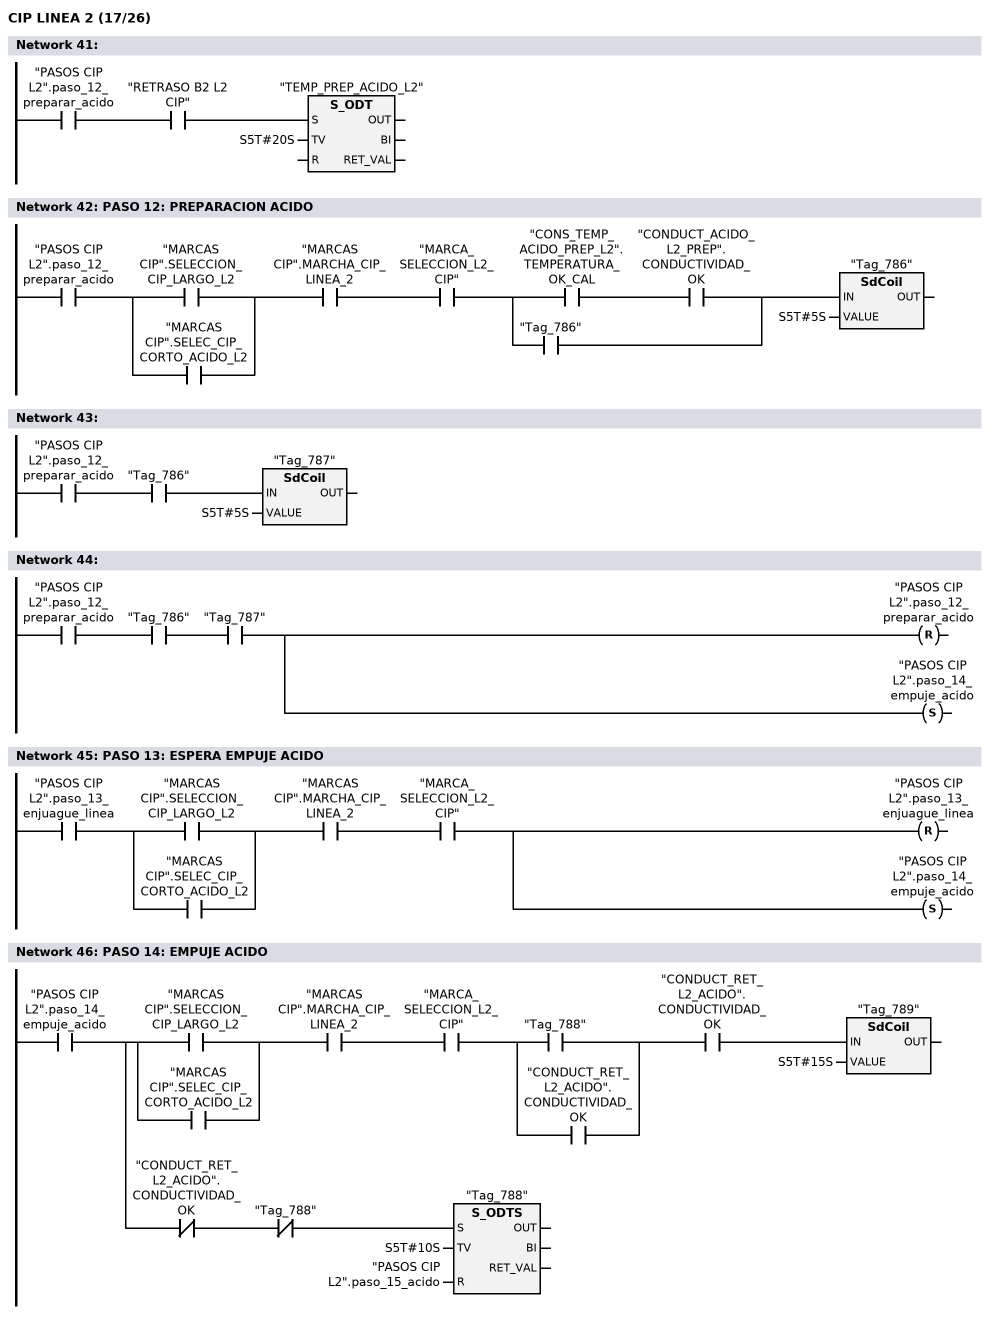
   RUNG wire#powerrail
      Contact( "PASOS CIP L2".paso_12_preparar_acido )
      Contact( "RETRASO B2 L2 CIP" )
      S_ODT(T_NO := "TEMP_PREP_ACIDO_L2", TV := S5T#20S, R :=, BI =>, RET_VAL =>)
   END_RUNG
   // the same network as SCL:
   #_s5time1 := S_ODT(T_NO := "TEMP_PREP_ACIDO_L2",
                      TV := S5T#20S,
                      S := "PASOS CIP L2".paso_12_preparar_acido AND "RETRASO B2 L2 CIP");
END_REGION

REGION Network 42: PASO 12: PREPARACION ACIDO
   // no SCL statement known for SdCoil: written as a call
   SdCoil(value := S5T#5S,
          in := "PASOS CIP L2".paso_12_preparar_acido AND ("MARCAS CIP".SELECCION_CIP_LARGO_L2 OR "MARCAS CIP".SELEC_CIP_CORTO_ACIDO_L2) AND "MARCAS CIP".MARCHA_CIP_LINEA_2 AND "MARCA_SELECCION_L2_CIP" AND (("CONS_TEMP_ACIDO_PREP_L2".TEMPERATURA_OK_CAL AND "CONDUCT_ACIDO_L2_PREP".CONDUCTIVIDAD_OK) OR "Tag_786"),
          operand := "Tag_786");
END_REGION

REGION Network 43
   // no SCL statement known for SdCoil: written as a call
   SdCoil(value := S5T#5S, operand := "Tag_787", in := "PASOS CIP L2".paso_12_preparar_acido AND "Tag_786");
END_REGION

REGION Network 44
   RUNG wire#powerrail
      Contact( "PASOS CIP L2".paso_12_preparar_acido )
      Contact( "Tag_786" )
      Contact( "Tag_787" )
      wire#w1
      R_Coil( "PASOS CIP L2".paso_12_preparar_acido )
   END_RUNG
   RUNG wire#w1
      S_Coil( "PASOS CIP L2".paso_14_empuje_acido )
   END_RUNG
   // the same network as SCL:
   #_w1 := "PASOS CIP L2".paso_12_preparar_acido AND "Tag_786" AND "Tag_787";
   IF #_w1 THEN
       "PASOS CIP L2".paso_12_preparar_acido := FALSE;
       "PASOS CIP L2".paso_14_empuje_acido := TRUE;
   END_IF;
END_REGION

REGION Network 45: PASO 13: ESPERA EMPUJE ACIDO
   RUNG wire#powerrail
      Contact( "PASOS CIP L2".paso_13_enjuague_linea )
      wire#w1
      Contact( "MARCAS CIP".SELECCION_CIP_LARGO_L2 )
      wire#w2
      Contact( "MARCAS CIP".MARCHA_CIP_LINEA_2 )
      Contact( "MARCA_SELECCION_L2_CIP" )
      wire#w3
      R_Coil( "PASOS CIP L2".paso_13_enjuague_linea )
   END_RUNG
   RUNG wire#w1
      Contact( "MARCAS CIP".SELEC_CIP_CORTO_ACIDO_L2 )
   END_RUNG wire#w2
   RUNG wire#w3
      S_Coil( "PASOS CIP L2".paso_14_empuje_acido )
   END_RUNG
   // the same network as SCL:
   #_w1 := "PASOS CIP L2".paso_13_enjuague_linea AND ("MARCAS CIP".SELECCION_CIP_LARGO_L2 OR "MARCAS CIP".SELEC_CIP_CORTO_ACIDO_L2) AND "MARCAS CIP".MARCHA_CIP_LINEA_2 AND "MARCA_SELECCION_L2_CIP";
   IF #_w1 THEN
       "PASOS CIP L2".paso_13_enjuague_linea := FALSE;
       "PASOS CIP L2".paso_14_empuje_acido := TRUE;
   END_IF;
END_REGION

REGION Network 46: PASO 14: EMPUJE ACIDO
   // no SCL statement known for SdCoil: written as a call
   #_w1 := "PASOS CIP L2".paso_14_empuje_acido;
   SdCoil(value := S5T#15S,
          operand := "Tag_789",
          in := "PASOS CIP L2".paso_14_empuje_acido AND ("MARCAS CIP".SELECCION_CIP_LARGO_L2 OR "MARCAS CIP".SELEC_CIP_CORTO_ACIDO_L2) AND "MARCAS CIP".MARCHA_CIP_LINEA_2 AND "MARCA_SELECCION_L2_CIP" AND ("Tag_788" OR "CONDUCT_RET_L2_ACIDO".CONDUCTIVIDAD_OK) AND "CONDUCT_RET_L2_ACIDO".CONDUCTIVIDAD_OK);
   #_s5time1 := S_ODTS(T_NO := "Tag_788",
                       TV := S5T#10S,
                       R := "PASOS CIP L2".paso_15_acido,
                       S := #_w1 AND NOT "CONDUCT_RET_L2_ACIDO".CONDUCTIVIDAD_OK AND NOT "Tag_788");
END_REGION

REGION Network 47
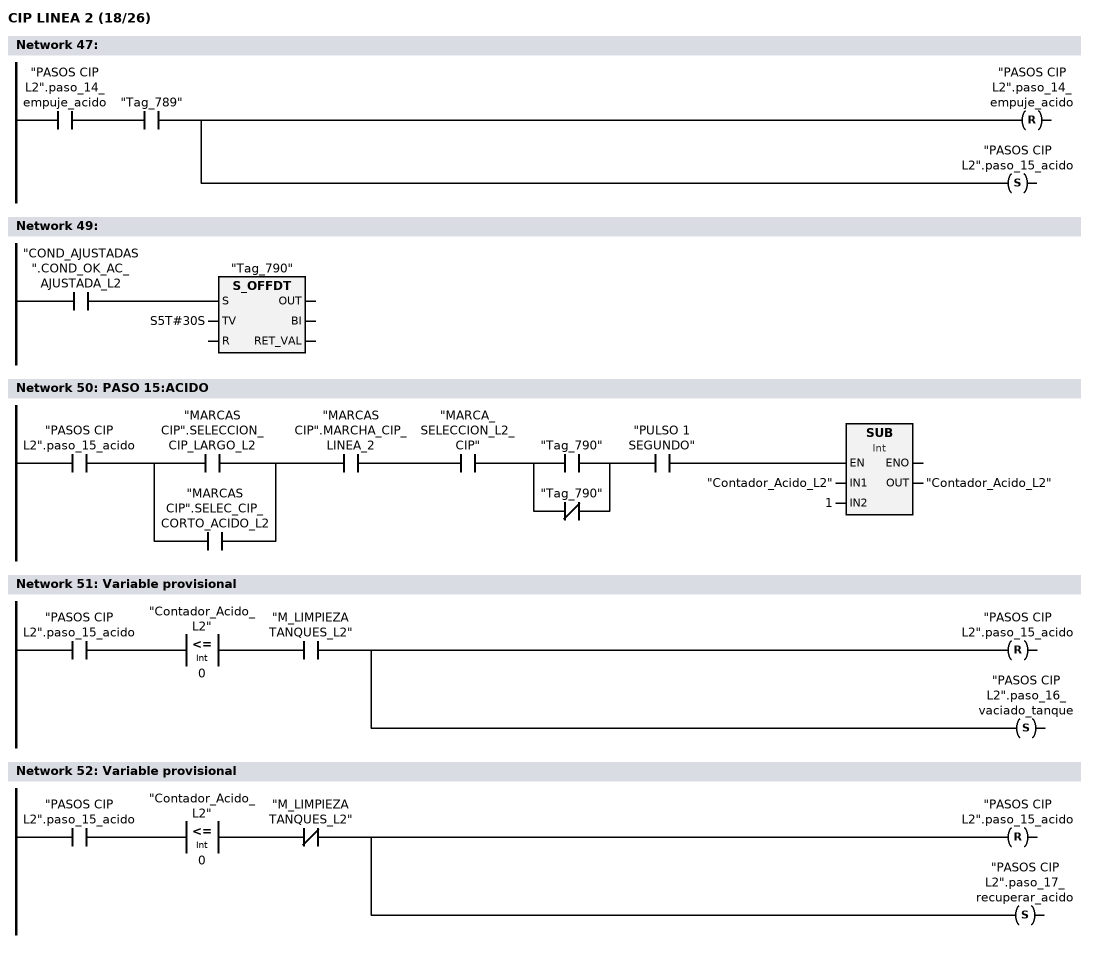
   RUNG wire#powerrail
      Contact( "PASOS CIP L2".paso_14_empuje_acido )
      Contact( "Tag_789" )
      wire#w1
      R_Coil( "PASOS CIP L2".paso_14_empuje_acido )
   END_RUNG
   RUNG wire#w1
      S_Coil( "PASOS CIP L2".paso_15_acido )
   END_RUNG
   // the same network as SCL:
   #_w1 := "PASOS CIP L2".paso_14_empuje_acido AND "Tag_789";
   IF #_w1 THEN
       "PASOS CIP L2".paso_14_empuje_acido := FALSE;
       "PASOS CIP L2".paso_15_acido := TRUE;
   END_IF;
END_REGION

NETWORK
TITLE = 
      A     "PASOS CIP L2".paso_15_acido;
      JC    c2;
      L     "SP TIM L2 CIP".TIM_PASO_15_L2;
      L     60;
      *I;
      T     "Contador_Acido_L2";
c2:   NOP   0;

REGION Network 49
   RUNG wire#powerrail
      Contact( "COND_AJUSTADAS".COND_OK_AC_AJUSTADA_L2 )
      S_OFFDT(T_NO := "Tag_790", TV := S5T#30S, R :=, BI =>, RET_VAL =>)
   END_RUNG
   // the same network as SCL:
   #_s5time1 := S_OFFDT(T_NO := "Tag_790", TV := S5T#30S, S := "COND_AJUSTADAS".COND_OK_AC_AJUSTADA_L2);
END_REGION

REGION Network 50: PASO 15:ACIDO
   RUNG wire#powerrail
      Contact( "PASOS CIP L2".paso_15_acido )
      wire#w1
      Contact( "MARCAS CIP".SELECCION_CIP_LARGO_L2 )
      wire#w2
      Contact( "MARCAS CIP".MARCHA_CIP_LINEA_2 )
      Contact( "MARCA_SELECCION_L2_CIP" )
      wire#w3
      Contact( "Tag_790" )
      wire#w4
      Contact( "PULSO 1 SEGUNDO" )
      { S7_Templates := "SrcType := Int"; S7_GenerateENO := "TRUE" } Sub(in1 := "Contador_Acido_L2", in2 := 1, out => "Contador_Acido_L2")
   END_RUNG
   RUNG wire#w1
      Contact( "MARCAS CIP".SELEC_CIP_CORTO_ACIDO_L2 )
   END_RUNG wire#w2
   RUNG wire#w3
      I_Contact( "Tag_790" )
   END_RUNG wire#w4
   // the same network as SCL:
   IF "PASOS CIP L2".paso_15_acido AND ("MARCAS CIP".SELECCION_CIP_LARGO_L2 OR "MARCAS CIP".SELEC_CIP_CORTO_ACIDO_L2) AND "MARCAS CIP".MARCHA_CIP_LINEA_2 AND "MARCA_SELECCION_L2_CIP" AND ("Tag_790" OR NOT "Tag_790") AND "PULSO 1 SEGUNDO" THEN
       "Contador_Acido_L2" := "Contador_Acido_L2" - 1;
   END_IF;
END_REGION

REGION Network 51: Variable provisional
   RUNG wire#powerrail
      Contact( "PASOS CIP L2".paso_15_acido )
      { S7_Templates := "SrcType := Int" } LE_Contact(in1 := "Contador_Acido_L2", in2 := 0)
      Contact( "M_LIMPIEZA TANQUES_L2" )
      wire#w1
      R_Coil( "PASOS CIP L2".paso_15_acido )
   END_RUNG
   RUNG wire#w1
      S_Coil( "PASOS CIP L2".paso_16_vaciado_tanque )
   END_RUNG
   // the same network as SCL:
   #_w1 := "PASOS CIP L2".paso_15_acido AND ("Contador_Acido_L2" <= 0) AND "M_LIMPIEZA TANQUES_L2";
   IF #_w1 THEN
       "PASOS CIP L2".paso_15_acido := FALSE;
       "PASOS CIP L2".paso_16_vaciado_tanque := TRUE;
   END_IF;
END_REGION

REGION Network 52: Variable provisional
   RUNG wire#powerrail
      Contact( "PASOS CIP L2".paso_15_acido )
      { S7_Templates := "SrcType := Int" } LE_Contact(in1 := "Contador_Acido_L2", in2 := 0)
      I_Contact( "M_LIMPIEZA TANQUES_L2" )
      wire#w1
      R_Coil( "PASOS CIP L2".paso_15_acido )
   END_RUNG
   RUNG wire#w1
      S_Coil( "PASOS CIP L2".paso_17_recuperar_acido )
   END_RUNG
   // the same network as SCL:
   #_w1 := "PASOS CIP L2".paso_15_acido AND ("Contador_Acido_L2" <= 0) AND NOT "M_LIMPIEZA TANQUES_L2";
   IF #_w1 THEN
       "PASOS CIP L2".paso_15_acido := FALSE;
       "PASOS CIP L2".paso_17_recuperar_acido := TRUE;
   END_IF;
END_REGION

REGION Network 53: PASO 16: VACIADO SI TANQUES
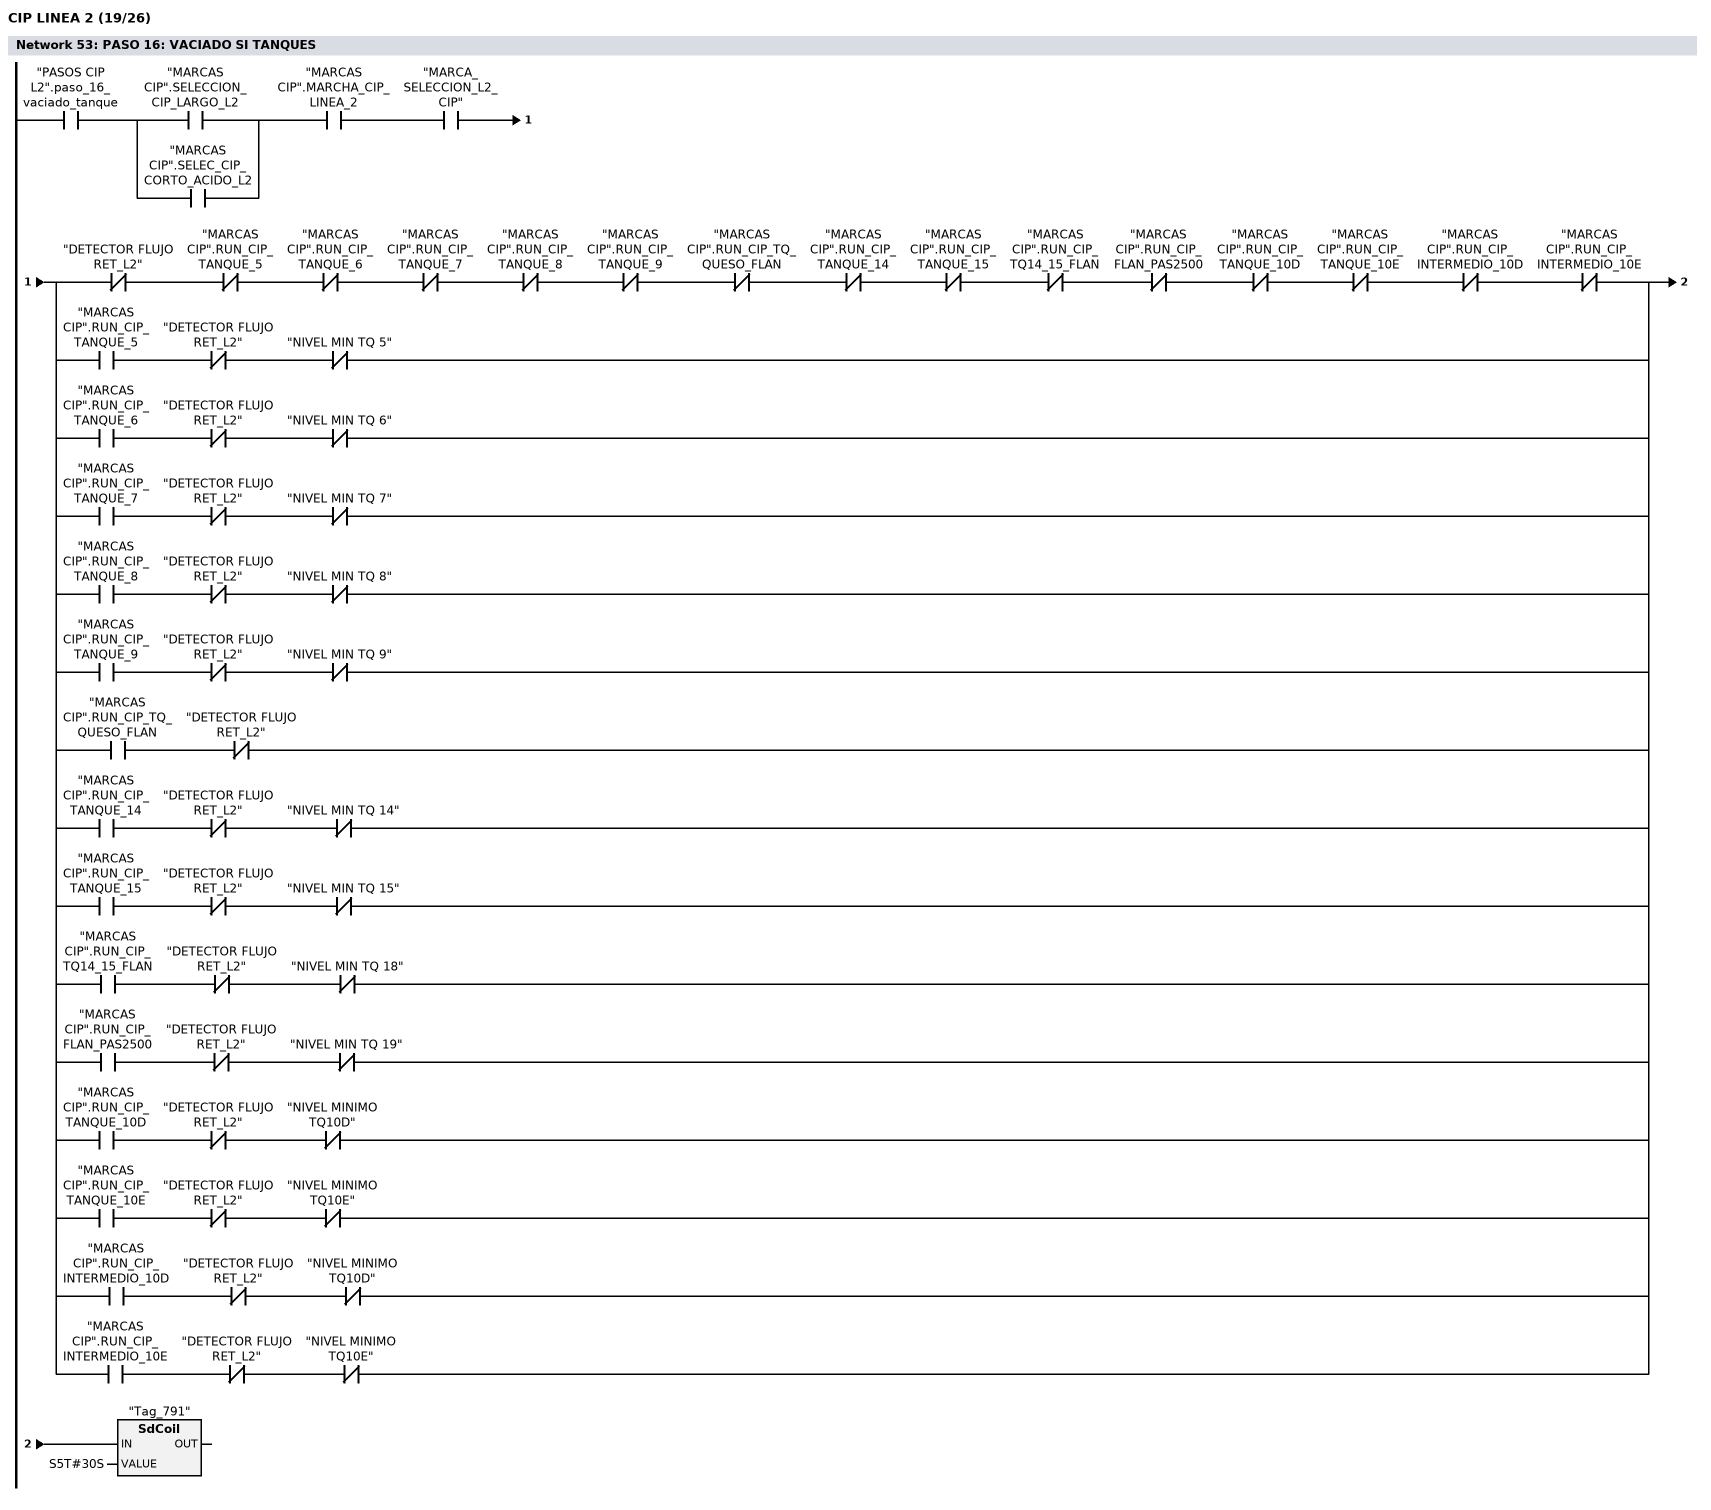
   // no SCL statement known for SdCoil: written as a call
   SdCoil(value := S5T#30S,
          in := "PASOS CIP L2".paso_16_vaciado_tanque AND ("MARCAS CIP".SELECCION_CIP_LARGO_L2 OR "MARCAS CIP".SELEC_CIP_CORTO_ACIDO_L2) AND "MARCAS CIP".MARCHA_CIP_LINEA_2 AND "MARCA_SELECCION_L2_CIP" AND ((NOT "DETECTOR FLUJO RET_L2" AND NOT "MARCAS CIP".RUN_CIP_TANQUE_5 AND NOT "MARCAS CIP".RUN_CIP_TANQUE_6 AND NOT "MARCAS CIP".RUN_CIP_TANQUE_7 AND NOT "MARCAS CIP".RUN_CIP_TANQUE_8 AND NOT "MARCAS CIP".RUN_CIP_TANQUE_9 AND NOT "MARCAS CIP".RUN_CIP_TQ_QUESO_FLAN AND NOT "MARCAS CIP".RUN_CIP_TANQUE_14 AND NOT "MARCAS CIP".RUN_CIP_TANQUE_15 AND NOT "MARCAS CIP".RUN_CIP_TQ14_15_FLAN AND NOT "MARCAS CIP".RUN_CIP_FLAN_PAS2500 AND NOT "MARCAS CIP".RUN_CIP_TANQUE_10D AND NOT "MARCAS CIP".RUN_CIP_TANQUE_10E AND NOT "MARCAS CIP".RUN_CIP_INTERMEDIO_10D AND NOT "MARCAS CIP".RUN_CIP_INTERMEDIO_10E) OR ("MARCAS CIP".RUN_CIP_TANQUE_5 AND NOT "DETECTOR FLUJO RET_L2" AND NOT "NIVEL MIN TQ 5") OR ("MARCAS CIP".RUN_CIP_TANQUE_6 AND NOT "DETECTOR FLUJO RET_L2" AND NOT "NIVEL MIN TQ 6") OR ("MARCAS CIP".RUN_CIP_TANQUE_7 AND NOT "DETECTOR FLUJO RET_L2" AND NOT "NIVEL MIN TQ 7") OR ("MARCAS CIP".RUN_CIP_TANQUE_8 AND NOT "DETECTOR FLUJO RET_L2" AND NOT "NIVEL MIN TQ 8") OR ("MARCAS CIP".RUN_CIP_TANQUE_9 AND NOT "DETECTOR FLUJO RET_L2" AND NOT "NIVEL MIN TQ 9") OR ("MARCAS CIP".RUN_CIP_TQ_QUESO_FLAN AND NOT "DETECTOR FLUJO RET_L2") OR ("MARCAS CIP".RUN_CIP_TANQUE_14 AND NOT "DETECTOR FLUJO RET_L2" AND NOT "NIVEL MIN TQ 14") OR ("MARCAS CIP".RUN_CIP_TANQUE_15 AND NOT "DETECTOR FLUJO RET_L2" AND NOT "NIVEL MIN TQ 15") OR ("MARCAS CIP".RUN_CIP_TQ14_15_FLAN AND NOT "DETECTOR FLUJO RET_L2" AND NOT "NIVEL MIN TQ 18") OR ("MARCAS CIP".RUN_CIP_FLAN_PAS2500 AND NOT "DETECTOR FLUJO RET_L2" AND NOT "NIVEL MIN TQ 19") OR ("MARCAS CIP".RUN_CIP_TANQUE_10D AND NOT "DETECTOR FLUJO RET_L2" AND NOT "NIVEL MINIMO TQ10D") OR ("MARCAS CIP".RUN_CIP_TANQUE_10E AND NOT "DETECTOR FLUJO RET_L2" AND NOT "NIVEL MINIMO TQ10E") OR ("MARCAS CIP".RUN_CIP_INTERMEDIO_10D AND NOT "DETECTOR FLUJO RET_L2" AND NOT "NIVEL MINIMO TQ10D") OR ("MARCAS CIP".RUN_CIP_INTERMEDIO_10E AND NOT "DETECTOR FLUJO RET_L2" AND NOT "NIVEL MINIMO TQ10E")),
          operand := "Tag_791");
END_REGION

REGION Network 54: Variable provisional
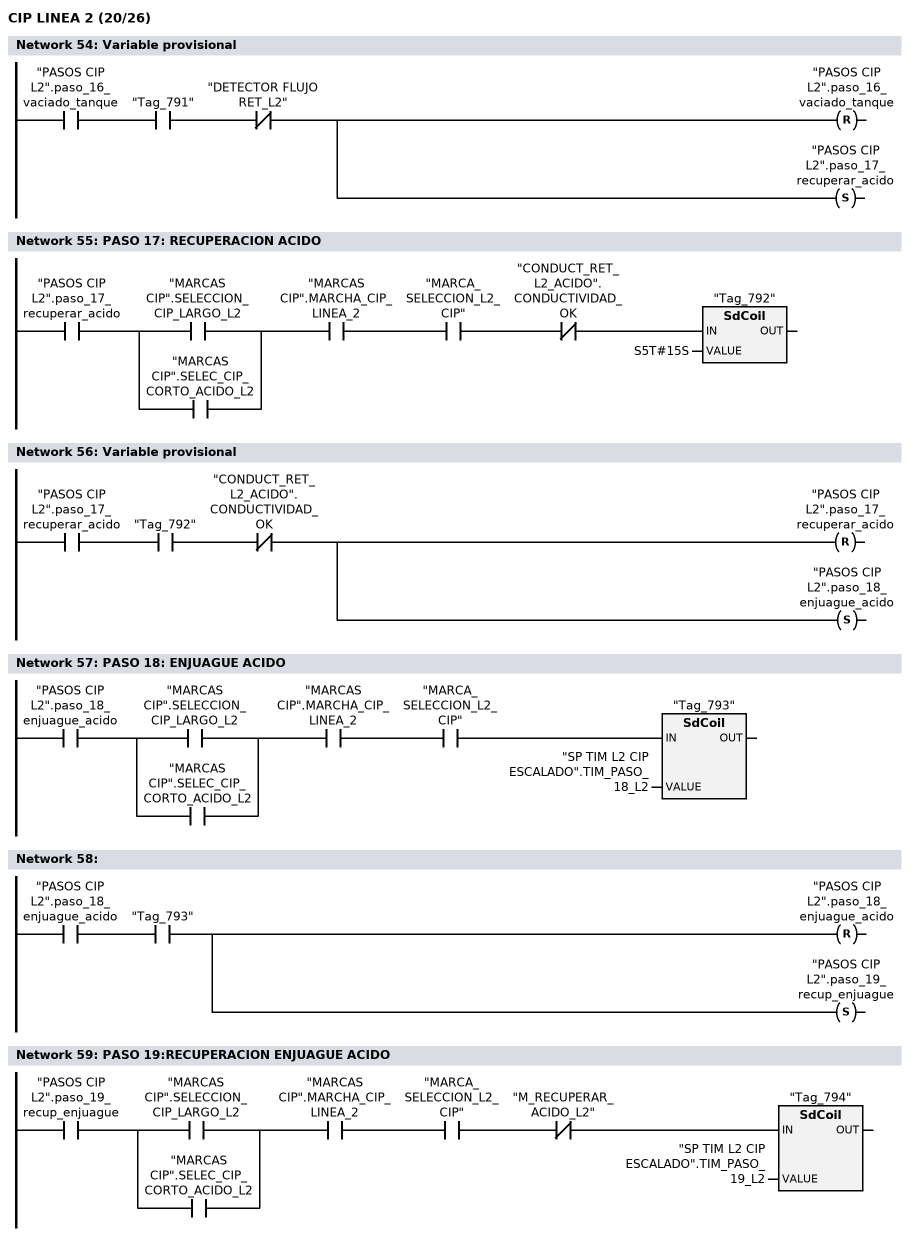
   RUNG wire#powerrail
      Contact( "PASOS CIP L2".paso_16_vaciado_tanque )
      Contact( "Tag_791" )
      I_Contact( "DETECTOR FLUJO RET_L2" )
      wire#w1
      R_Coil( "PASOS CIP L2".paso_16_vaciado_tanque )
   END_RUNG
   RUNG wire#w1
      S_Coil( "PASOS CIP L2".paso_17_recuperar_acido )
   END_RUNG
   // the same network as SCL:
   #_w1 := "PASOS CIP L2".paso_16_vaciado_tanque AND "Tag_791" AND NOT "DETECTOR FLUJO RET_L2";
   IF #_w1 THEN
       "PASOS CIP L2".paso_16_vaciado_tanque := FALSE;
       "PASOS CIP L2".paso_17_recuperar_acido := TRUE;
   END_IF;
END_REGION

REGION Network 55: PASO 17: RECUPERACION ACIDO
   // no SCL statement known for SdCoil: written as a call
   SdCoil(value := S5T#15S,
          operand := "Tag_792",
          in := "PASOS CIP L2".paso_17_recuperar_acido AND ("MARCAS CIP".SELECCION_CIP_LARGO_L2 OR "MARCAS CIP".SELEC_CIP_CORTO_ACIDO_L2) AND "MARCAS CIP".MARCHA_CIP_LINEA_2 AND "MARCA_SELECCION_L2_CIP" AND NOT "CONDUCT_RET_L2_ACIDO".CONDUCTIVIDAD_OK);
END_REGION

REGION Network 56: Variable provisional
   RUNG wire#powerrail
      Contact( "PASOS CIP L2".paso_17_recuperar_acido )
      Contact( "Tag_792" )
      I_Contact( "CONDUCT_RET_L2_ACIDO".CONDUCTIVIDAD_OK )
      wire#w1
      R_Coil( "PASOS CIP L2".paso_17_recuperar_acido )
   END_RUNG
   RUNG wire#w1
      S_Coil( "PASOS CIP L2".paso_18_enjuague_acido )
   END_RUNG
   // the same network as SCL:
   #_w1 := "PASOS CIP L2".paso_17_recuperar_acido AND "Tag_792" AND NOT "CONDUCT_RET_L2_ACIDO".CONDUCTIVIDAD_OK;
   IF #_w1 THEN
       "PASOS CIP L2".paso_17_recuperar_acido := FALSE;
       "PASOS CIP L2".paso_18_enjuague_acido := TRUE;
   END_IF;
END_REGION

REGION Network 57: PASO 18: ENJUAGUE ACIDO
   // no SCL statement known for SdCoil: written as a call
   SdCoil(value := "SP TIM L2 CIP ESCALADO".TIM_PASO_18_L2,
          operand := "Tag_793",
          in := "PASOS CIP L2".paso_18_enjuague_acido AND ("MARCAS CIP".SELECCION_CIP_LARGO_L2 OR "MARCAS CIP".SELEC_CIP_CORTO_ACIDO_L2) AND "MARCAS CIP".MARCHA_CIP_LINEA_2 AND "MARCA_SELECCION_L2_CIP");
END_REGION

REGION Network 58
   RUNG wire#powerrail
      Contact( "PASOS CIP L2".paso_18_enjuague_acido )
      Contact( "Tag_793" )
      wire#w1
      R_Coil( "PASOS CIP L2".paso_18_enjuague_acido )
   END_RUNG
   RUNG wire#w1
      S_Coil( "PASOS CIP L2".paso_19_recup_enjuague )
   END_RUNG
   // the same network as SCL:
   #_w1 := "PASOS CIP L2".paso_18_enjuague_acido AND "Tag_793";
   IF #_w1 THEN
       "PASOS CIP L2".paso_18_enjuague_acido := FALSE;
       "PASOS CIP L2".paso_19_recup_enjuague := TRUE;
   END_IF;
END_REGION

REGION Network 59: PASO 19:RECUPERACION ENJUAGUE ACIDO
   // no SCL statement known for SdCoil: written as a call
   SdCoil(value := "SP TIM L2 CIP ESCALADO".TIM_PASO_19_L2,
          operand := "Tag_794",
          in := "PASOS CIP L2".paso_19_recup_enjuague AND ("MARCAS CIP".SELECCION_CIP_LARGO_L2 OR "MARCAS CIP".SELEC_CIP_CORTO_ACIDO_L2) AND "MARCAS CIP".MARCHA_CIP_LINEA_2 AND "MARCA_SELECCION_L2_CIP" AND NOT "M_RECUPERAR_ACIDO_L2");
END_REGION

REGION Network 60
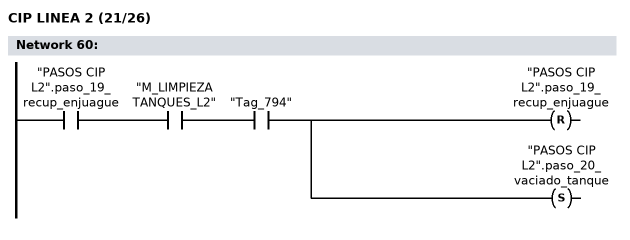
   RUNG wire#powerrail
      Contact( "PASOS CIP L2".paso_19_recup_enjuague )
      Contact( "M_LIMPIEZA TANQUES_L2" )
      Contact( "Tag_794" )
      wire#w1
      R_Coil( "PASOS CIP L2".paso_19_recup_enjuague )
   END_RUNG
   RUNG wire#w1
      S_Coil( "PASOS CIP L2".paso_20_vaciado_tanque )
   END_RUNG
   // the same network as SCL:
   #_w1 := "PASOS CIP L2".paso_19_recup_enjuague AND "M_LIMPIEZA TANQUES_L2" AND "Tag_794";
   IF #_w1 THEN
       "PASOS CIP L2".paso_19_recup_enjuague := FALSE;
       "PASOS CIP L2".paso_20_vaciado_tanque := TRUE;
   END_IF;
END_REGION

REGION Network 61
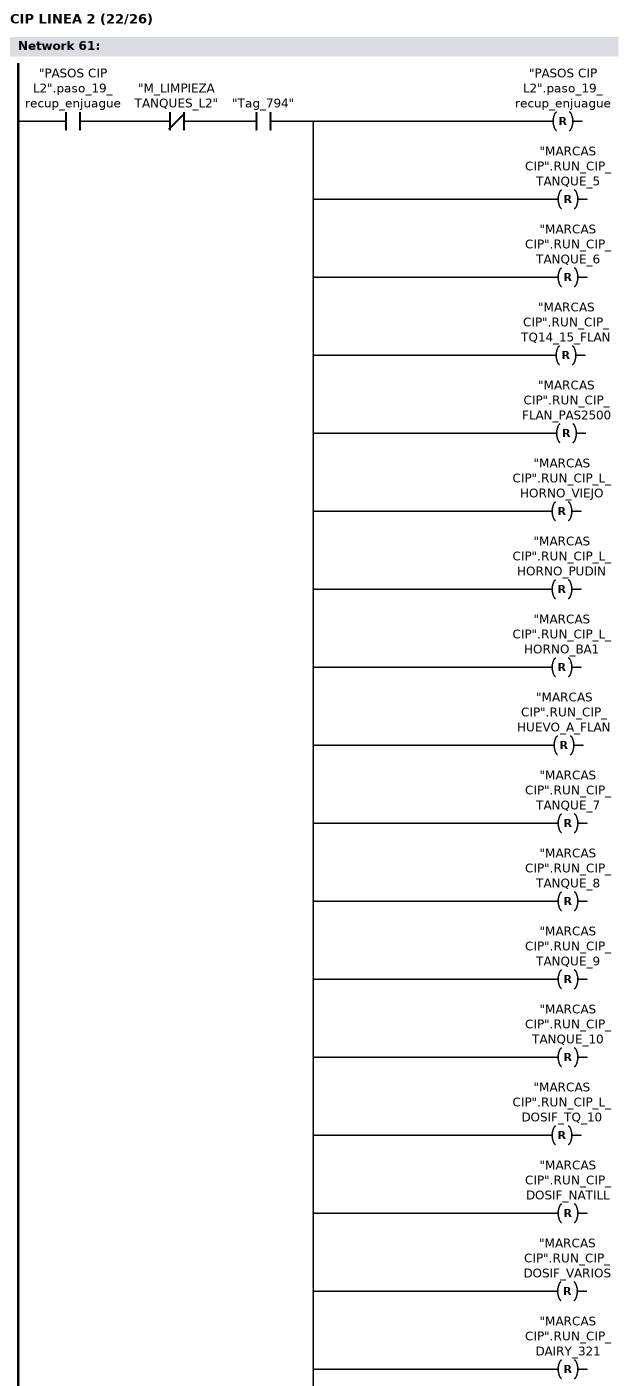
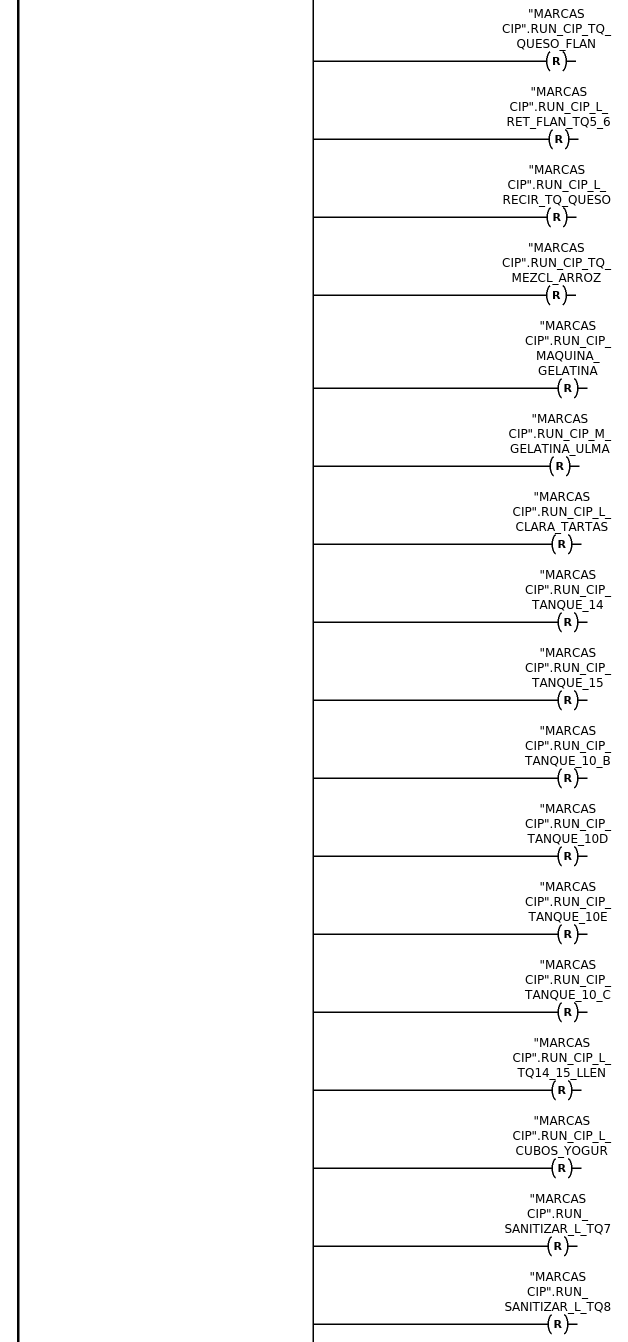
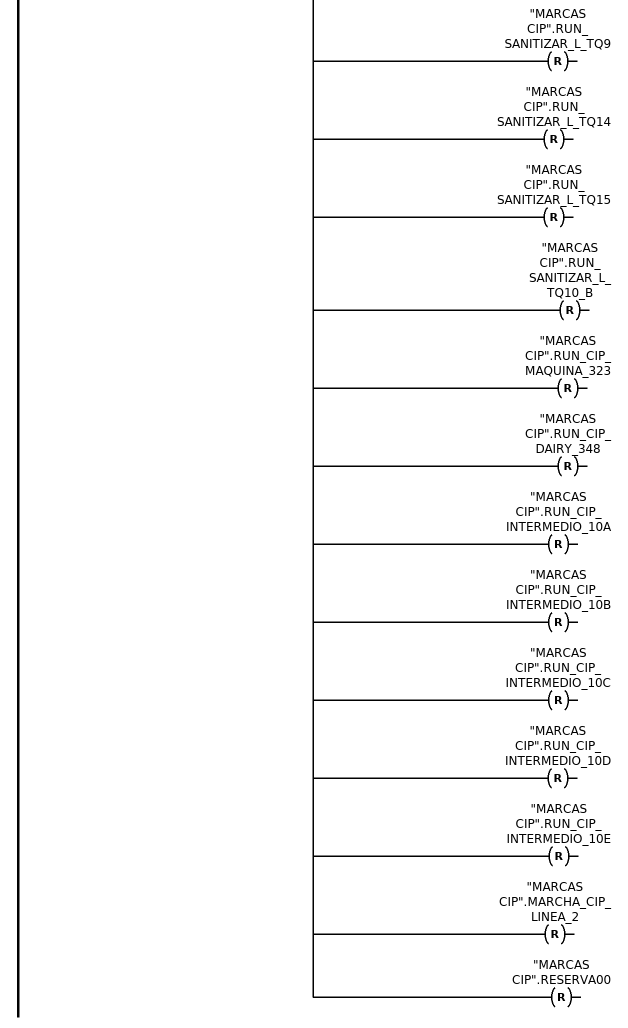
   RUNG wire#powerrail
      Contact( "PASOS CIP L2".paso_19_recup_enjuague )
      I_Contact( "M_LIMPIEZA TANQUES_L2" )
      Contact( "Tag_794" )
      wire#w1
      R_Coil( "PASOS CIP L2".paso_19_recup_enjuague )
   END_RUNG
   RUNG wire#w1
      R_Coil( "MARCAS CIP".RUN_CIP_TANQUE_5 )
   END_RUNG
   RUNG wire#w1
      R_Coil( "MARCAS CIP".RUN_CIP_TANQUE_6 )
   END_RUNG
   RUNG wire#w1
      R_Coil( "MARCAS CIP".RUN_CIP_TQ14_15_FLAN )
   END_RUNG
   RUNG wire#w1
      R_Coil( "MARCAS CIP".RUN_CIP_FLAN_PAS2500 )
   END_RUNG
   RUNG wire#w1
      R_Coil( "MARCAS CIP".RUN_CIP_L_HORNO_VIEJO )
   END_RUNG
   RUNG wire#w1
      R_Coil( "MARCAS CIP".RUN_CIP_L_HORNO_PUDIN )
   END_RUNG
   RUNG wire#w1
      R_Coil( "MARCAS CIP".RUN_CIP_L_HORNO_BA1 )
   END_RUNG
   RUNG wire#w1
      R_Coil( "MARCAS CIP".RUN_CIP_HUEVO_A_FLAN )
   END_RUNG
   RUNG wire#w1
      R_Coil( "MARCAS CIP".RUN_CIP_TANQUE_7 )
   END_RUNG
   RUNG wire#w1
      R_Coil( "MARCAS CIP".RUN_CIP_TANQUE_8 )
   END_RUNG
   RUNG wire#w1
      R_Coil( "MARCAS CIP".RUN_CIP_TANQUE_9 )
   END_RUNG
   RUNG wire#w1
      R_Coil( "MARCAS CIP".RUN_CIP_TANQUE_10 )
   END_RUNG
   RUNG wire#w1
      R_Coil( "MARCAS CIP".RUN_CIP_L_DOSIF_TQ_10 )
   END_RUNG
   RUNG wire#w1
      R_Coil( "MARCAS CIP".RUN_CIP_DOSIF_NATILL )
   END_RUNG
   RUNG wire#w1
      R_Coil( "MARCAS CIP".RUN_CIP_DOSIF_VARIOS )
   END_RUNG
   RUNG wire#w1
      R_Coil( "MARCAS CIP".RUN_CIP_DAIRY_321 )
   END_RUNG
   RUNG wire#w1
      R_Coil( "MARCAS CIP".RUN_CIP_TQ_QUESO_FLAN )
   END_RUNG
   RUNG wire#w1
      R_Coil( "MARCAS CIP".RUN_CIP_L_RET_FLAN_TQ5_6 )
   END_RUNG
   RUNG wire#w1
      R_Coil( "MARCAS CIP".RUN_CIP_L_RECIR_TQ_QUESO )
   END_RUNG
   RUNG wire#w1
      R_Coil( "MARCAS CIP".RUN_CIP_TQ_MEZCL_ARROZ )
   END_RUNG
   RUNG wire#w1
      R_Coil( "MARCAS CIP".RUN_CIP_MAQUINA_GELATINA )
   END_RUNG
   RUNG wire#w1
      R_Coil( "MARCAS CIP".RUN_CIP_M_GELATINA_ULMA )
   END_RUNG
   RUNG wire#w1
      R_Coil( "MARCAS CIP".RUN_CIP_L_CLARA_TARTAS )
   END_RUNG
   RUNG wire#w1
      R_Coil( "MARCAS CIP".RUN_CIP_TANQUE_14 )
   END_RUNG
   RUNG wire#w1
      R_Coil( "MARCAS CIP".RUN_CIP_TANQUE_15 )
   END_RUNG
   RUNG wire#w1
      R_Coil( "MARCAS CIP".RUN_CIP_TANQUE_10_B )
   END_RUNG
   RUNG wire#w1
      R_Coil( "MARCAS CIP".RUN_CIP_TANQUE_10D )
   END_RUNG
   RUNG wire#w1
      R_Coil( "MARCAS CIP".RUN_CIP_TANQUE_10E )
   END_RUNG
   RUNG wire#w1
      R_Coil( "MARCAS CIP".RUN_CIP_TANQUE_10_C )
   END_RUNG
   RUNG wire#w1
      R_Coil( "MARCAS CIP".RUN_CIP_L_TQ14_15_LLEN )
   END_RUNG
   RUNG wire#w1
      R_Coil( "MARCAS CIP".RUN_CIP_L_CUBOS_YOGUR )
   END_RUNG
   RUNG wire#w1
      R_Coil( "MARCAS CIP".RUN_SANITIZAR_L_TQ7 )
   END_RUNG
   RUNG wire#w1
      R_Coil( "MARCAS CIP".RUN_SANITIZAR_L_TQ8 )
   END_RUNG
   RUNG wire#w1
      R_Coil( "MARCAS CIP".RUN_SANITIZAR_L_TQ9 )
   END_RUNG
   RUNG wire#w1
      R_Coil( "MARCAS CIP".RUN_SANITIZAR_L_TQ14 )
   END_RUNG
   RUNG wire#w1
      R_Coil( "MARCAS CIP".RUN_SANITIZAR_L_TQ15 )
   END_RUNG
   RUNG wire#w1
      R_Coil( "MARCAS CIP".RUN_SANITIZAR_L_TQ10_B )
   END_RUNG
   RUNG wire#w1
      R_Coil( "MARCAS CIP".RUN_CIP_MAQUINA_323 )
   END_RUNG
   RUNG wire#w1
      R_Coil( "MARCAS CIP".RUN_CIP_DAIRY_348 )
   END_RUNG
   RUNG wire#w1
      R_Coil( "MARCAS CIP".RUN_CIP_INTERMEDIO_10A )
   END_RUNG
   RUNG wire#w1
      R_Coil( "MARCAS CIP".RUN_CIP_INTERMEDIO_10B )
   END_RUNG
   RUNG wire#w1
      R_Coil( "MARCAS CIP".RUN_CIP_INTERMEDIO_10C )
   END_RUNG
   RUNG wire#w1
      R_Coil( "MARCAS CIP".RUN_CIP_INTERMEDIO_10D )
   END_RUNG
   RUNG wire#w1
      R_Coil( "MARCAS CIP".RUN_CIP_INTERMEDIO_10E )
   END_RUNG
   RUNG wire#w1
      R_Coil( "MARCAS CIP".MARCHA_CIP_LINEA_2 )
   END_RUNG
   RUNG wire#w1
      R_Coil( "MARCAS CIP".RESERVA00 )
   END_RUNG
   // the same network as SCL:
   #_w1 := "PASOS CIP L2".paso_19_recup_enjuague AND NOT "M_LIMPIEZA TANQUES_L2" AND "Tag_794";
   IF #_w1 THEN
       "PASOS CIP L2".paso_19_recup_enjuague := FALSE;
       "MARCAS CIP".RUN_CIP_TANQUE_5 := FALSE;
       "MARCAS CIP".RUN_CIP_TANQUE_6 := FALSE;
       "MARCAS CIP".RUN_CIP_TQ14_15_FLAN := FALSE;
       "MARCAS CIP".RUN_CIP_FLAN_PAS2500 := FALSE;
       "MARCAS CIP".RUN_CIP_L_HORNO_VIEJO := FALSE;
       "MARCAS CIP".RUN_CIP_L_HORNO_PUDIN := FALSE;
       "MARCAS CIP".RUN_CIP_L_HORNO_BA1 := FALSE;
       "MARCAS CIP".RUN_CIP_HUEVO_A_FLAN := FALSE;
       "MARCAS CIP".RUN_CIP_TANQUE_7 := FALSE;
       "MARCAS CIP".RUN_CIP_TANQUE_8 := FALSE;
       "MARCAS CIP".RUN_CIP_TANQUE_9 := FALSE;
       "MARCAS CIP".RUN_CIP_TANQUE_10 := FALSE;
       "MARCAS CIP".RUN_CIP_L_DOSIF_TQ_10 := FALSE;
       "MARCAS CIP".RUN_CIP_DOSIF_NATILL := FALSE;
       "MARCAS CIP".RUN_CIP_DOSIF_VARIOS := FALSE;
       "MARCAS CIP".RUN_CIP_DAIRY_321 := FALSE;
       "MARCAS CIP".RUN_CIP_TQ_QUESO_FLAN := FALSE;
       "MARCAS CIP".RUN_CIP_L_RET_FLAN_TQ5_6 := FALSE;
       "MARCAS CIP".RUN_CIP_L_RECIR_TQ_QUESO := FALSE;
       "MARCAS CIP".RUN_CIP_TQ_MEZCL_ARROZ := FALSE;
       "MARCAS CIP".RUN_CIP_MAQUINA_GELATINA := FALSE;
       "MARCAS CIP".RUN_CIP_M_GELATINA_ULMA := FALSE;
       "MARCAS CIP".RUN_CIP_L_CLARA_TARTAS := FALSE;
       "MARCAS CIP".RUN_CIP_TANQUE_14 := FALSE;
       "MARCAS CIP".RUN_CIP_TANQUE_15 := FALSE;
       "MARCAS CIP".RUN_CIP_TANQUE_10_B := FALSE;
       "MARCAS CIP".RUN_CIP_TANQUE_10D := FALSE;
       "MARCAS CIP".RUN_CIP_TANQUE_10E := FALSE;
       "MARCAS CIP".RUN_CIP_TANQUE_10_C := FALSE;
       "MARCAS CIP".RUN_CIP_L_TQ14_15_LLEN := FALSE;
       "MARCAS CIP".RUN_CIP_L_CUBOS_YOGUR := FALSE;
       "MARCAS CIP".RUN_SANITIZAR_L_TQ7 := FALSE;
       "MARCAS CIP".RUN_SANITIZAR_L_TQ8 := FALSE;
       "MARCAS CIP".RUN_SANITIZAR_L_TQ9 := FALSE;
       "MARCAS CIP".RUN_SANITIZAR_L_TQ14 := FALSE;
       "MARCAS CIP".RUN_SANITIZAR_L_TQ15 := FALSE;
       "MARCAS CIP".RUN_SANITIZAR_L_TQ10_B := FALSE;
       "MARCAS CIP".RUN_CIP_MAQUINA_323 := FALSE;
       "MARCAS CIP".RUN_CIP_DAIRY_348 := FALSE;
       "MARCAS CIP".RUN_CIP_INTERMEDIO_10A := FALSE;
       "MARCAS CIP".RUN_CIP_INTERMEDIO_10B := FALSE;
       "MARCAS CIP".RUN_CIP_INTERMEDIO_10C := FALSE;
       "MARCAS CIP".RUN_CIP_INTERMEDIO_10D := FALSE;
       "MARCAS CIP".RUN_CIP_INTERMEDIO_10E := FALSE;
       "MARCAS CIP".MARCHA_CIP_LINEA_2 := FALSE;
       "MARCAS CIP".RESERVA00 := FALSE;
   END_IF;
END_REGION

REGION Network 62: PASO 19: VACIADO SI TANQUES
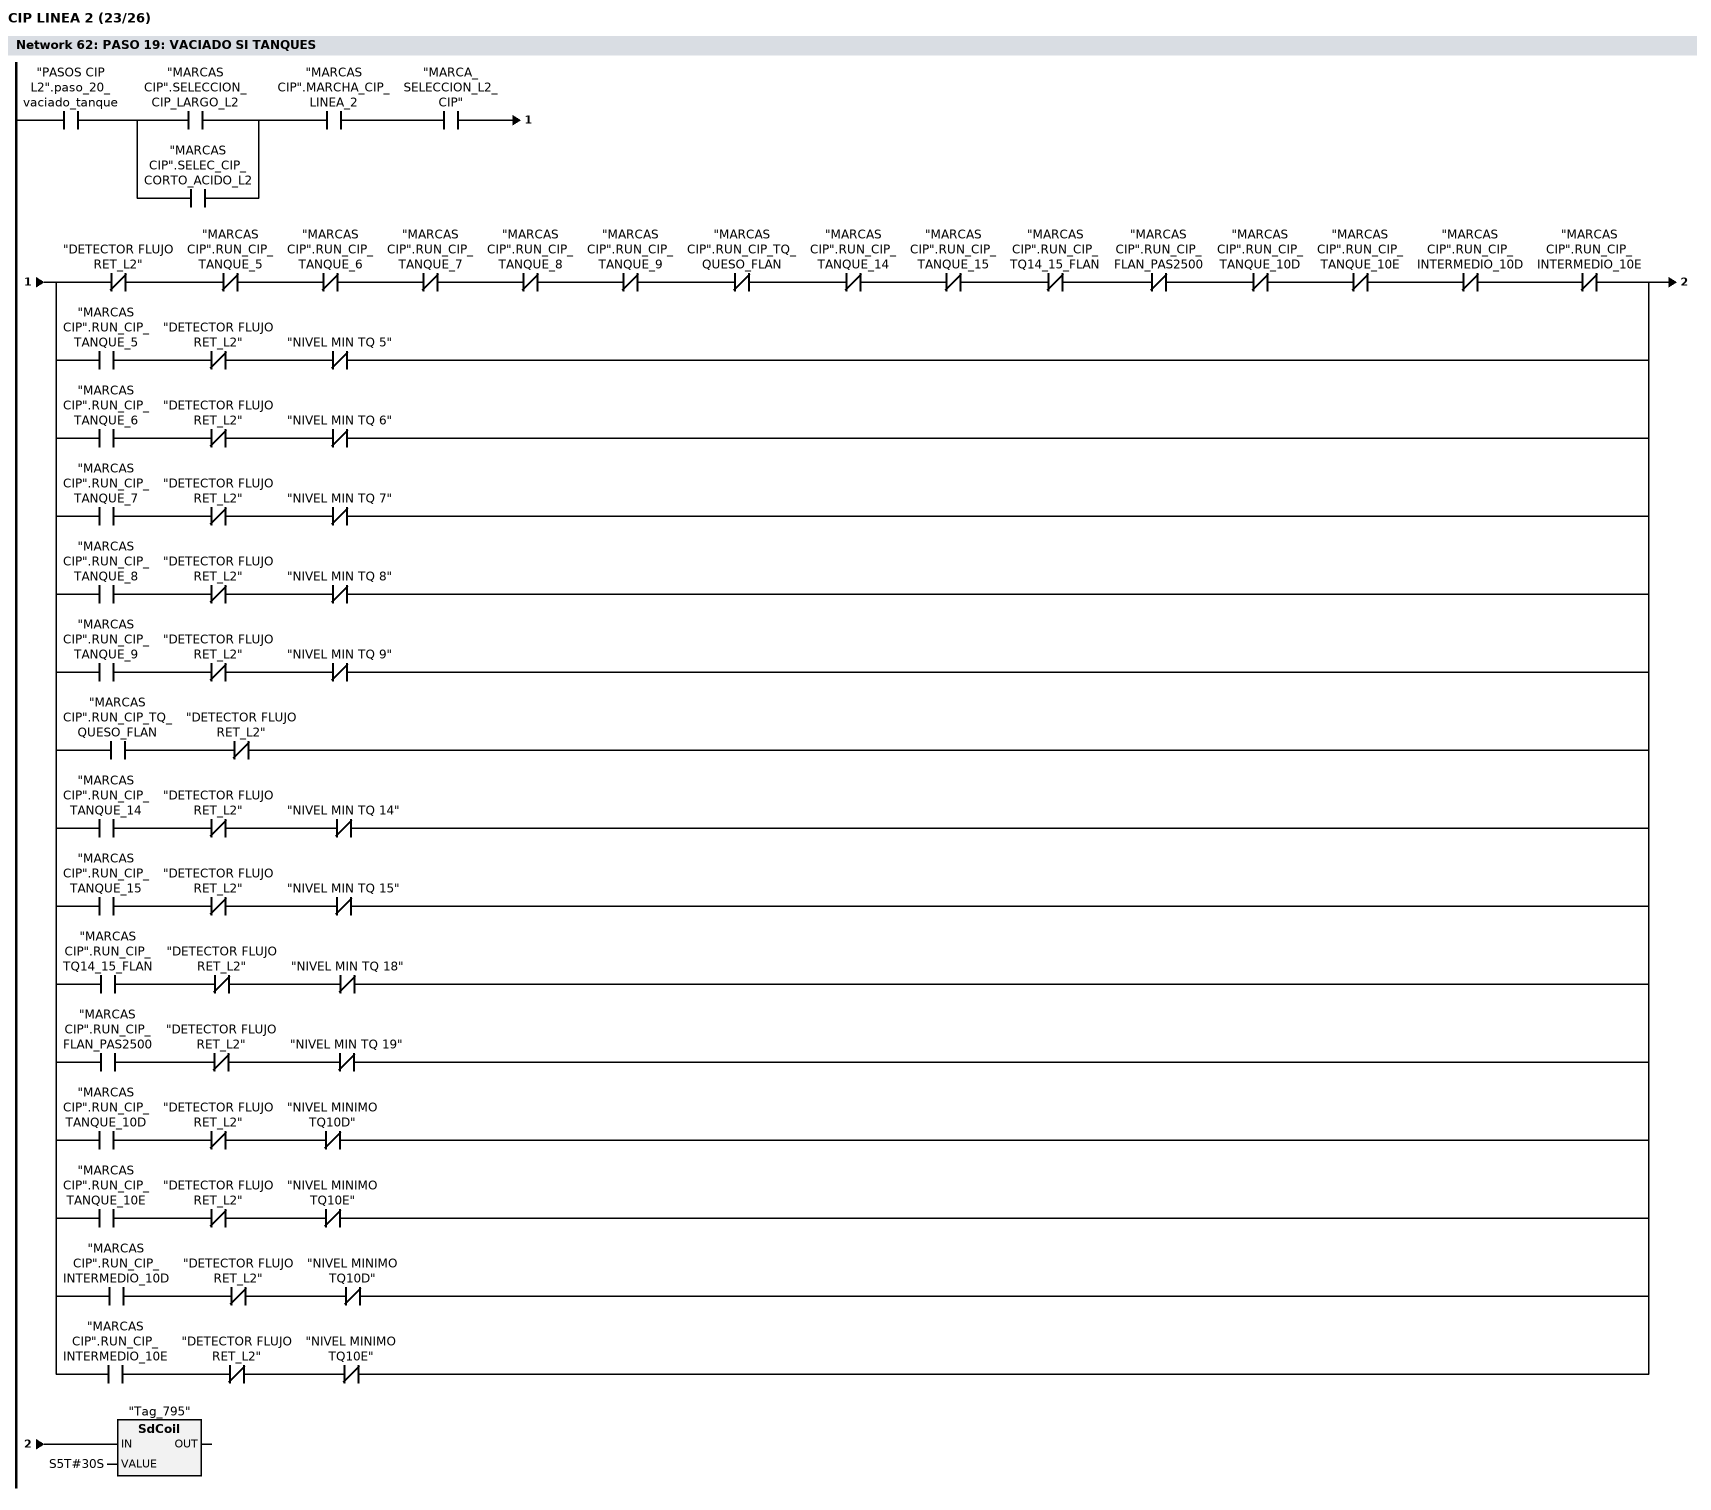
   // no SCL statement known for SdCoil: written as a call
   SdCoil(value := S5T#30S,
          in := "PASOS CIP L2".paso_20_vaciado_tanque AND ("MARCAS CIP".SELECCION_CIP_LARGO_L2 OR "MARCAS CIP".SELEC_CIP_CORTO_ACIDO_L2) AND "MARCAS CIP".MARCHA_CIP_LINEA_2 AND "MARCA_SELECCION_L2_CIP" AND ((NOT "DETECTOR FLUJO RET_L2" AND NOT "MARCAS CIP".RUN_CIP_TANQUE_5 AND NOT "MARCAS CIP".RUN_CIP_TANQUE_6 AND NOT "MARCAS CIP".RUN_CIP_TANQUE_7 AND NOT "MARCAS CIP".RUN_CIP_TANQUE_8 AND NOT "MARCAS CIP".RUN_CIP_TANQUE_9 AND NOT "MARCAS CIP".RUN_CIP_TQ_QUESO_FLAN AND NOT "MARCAS CIP".RUN_CIP_TANQUE_14 AND NOT "MARCAS CIP".RUN_CIP_TANQUE_15 AND NOT "MARCAS CIP".RUN_CIP_TQ14_15_FLAN AND NOT "MARCAS CIP".RUN_CIP_FLAN_PAS2500 AND NOT "MARCAS CIP".RUN_CIP_TANQUE_10D AND NOT "MARCAS CIP".RUN_CIP_TANQUE_10E AND NOT "MARCAS CIP".RUN_CIP_INTERMEDIO_10D AND NOT "MARCAS CIP".RUN_CIP_INTERMEDIO_10E) OR ("MARCAS CIP".RUN_CIP_TANQUE_5 AND NOT "DETECTOR FLUJO RET_L2" AND NOT "NIVEL MIN TQ 5") OR ("MARCAS CIP".RUN_CIP_TANQUE_6 AND NOT "DETECTOR FLUJO RET_L2" AND NOT "NIVEL MIN TQ 6") OR ("MARCAS CIP".RUN_CIP_TANQUE_7 AND NOT "DETECTOR FLUJO RET_L2" AND NOT "NIVEL MIN TQ 7") OR ("MARCAS CIP".RUN_CIP_TANQUE_8 AND NOT "DETECTOR FLUJO RET_L2" AND NOT "NIVEL MIN TQ 8") OR ("MARCAS CIP".RUN_CIP_TANQUE_9 AND NOT "DETECTOR FLUJO RET_L2" AND NOT "NIVEL MIN TQ 9") OR ("MARCAS CIP".RUN_CIP_TQ_QUESO_FLAN AND NOT "DETECTOR FLUJO RET_L2") OR ("MARCAS CIP".RUN_CIP_TANQUE_14 AND NOT "DETECTOR FLUJO RET_L2" AND NOT "NIVEL MIN TQ 14") OR ("MARCAS CIP".RUN_CIP_TANQUE_15 AND NOT "DETECTOR FLUJO RET_L2" AND NOT "NIVEL MIN TQ 15") OR ("MARCAS CIP".RUN_CIP_TQ14_15_FLAN AND NOT "DETECTOR FLUJO RET_L2" AND NOT "NIVEL MIN TQ 18") OR ("MARCAS CIP".RUN_CIP_FLAN_PAS2500 AND NOT "DETECTOR FLUJO RET_L2" AND NOT "NIVEL MIN TQ 19") OR ("MARCAS CIP".RUN_CIP_TANQUE_10D AND NOT "DETECTOR FLUJO RET_L2" AND NOT "NIVEL MINIMO TQ10D") OR ("MARCAS CIP".RUN_CIP_TANQUE_10E AND NOT "DETECTOR FLUJO RET_L2" AND NOT "NIVEL MINIMO TQ10E") OR ("MARCAS CIP".RUN_CIP_INTERMEDIO_10D AND NOT "DETECTOR FLUJO RET_L2" AND NOT "NIVEL MINIMO TQ10D") OR ("MARCAS CIP".RUN_CIP_INTERMEDIO_10E AND NOT "DETECTOR FLUJO RET_L2" AND NOT "NIVEL MINIMO TQ10E")),
          operand := "Tag_795");
END_REGION

REGION Network 63: FIN DE CICLO
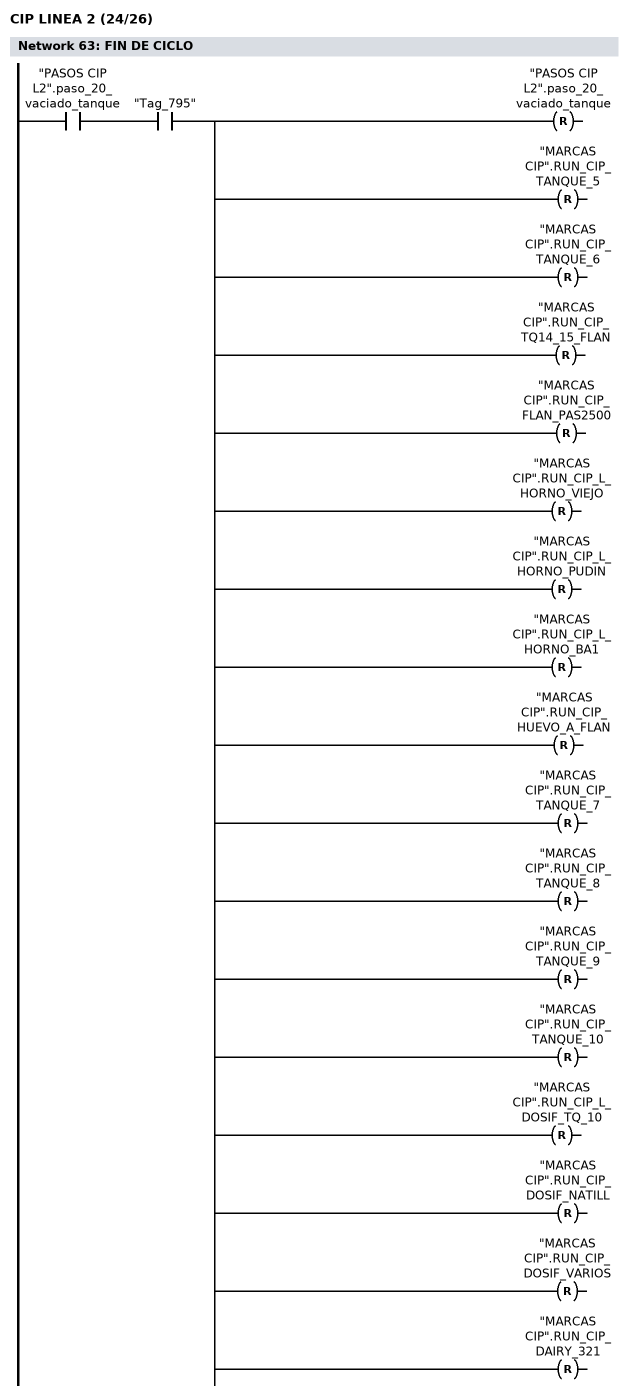
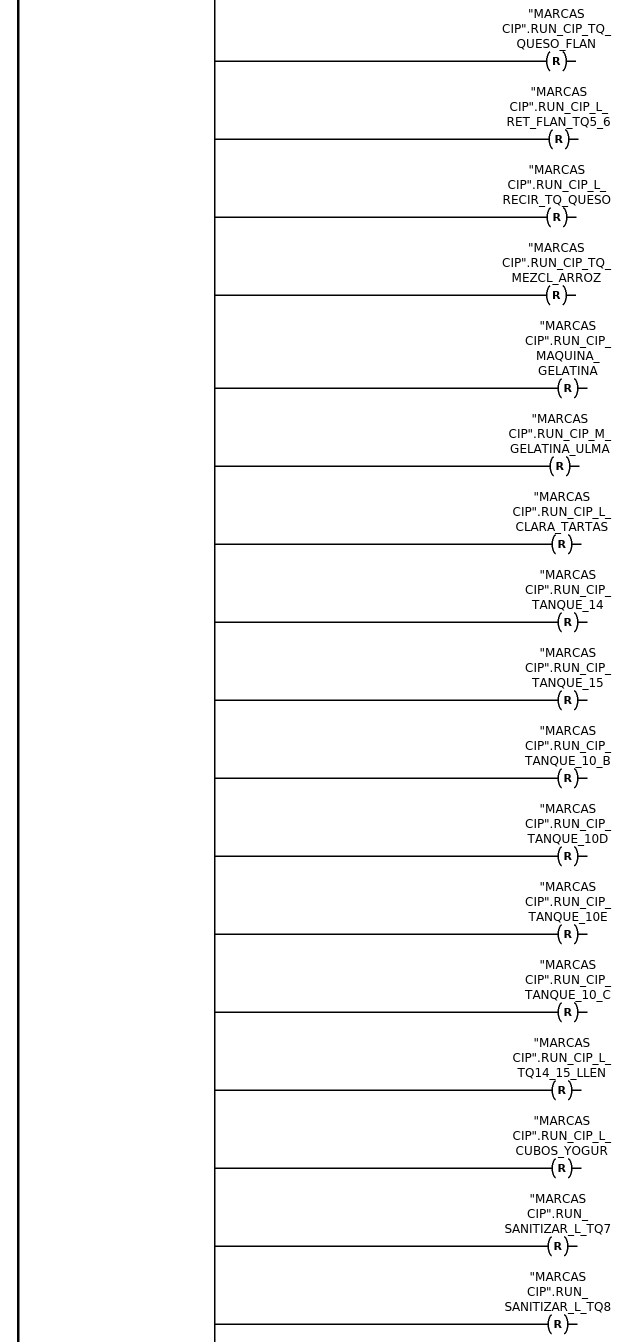
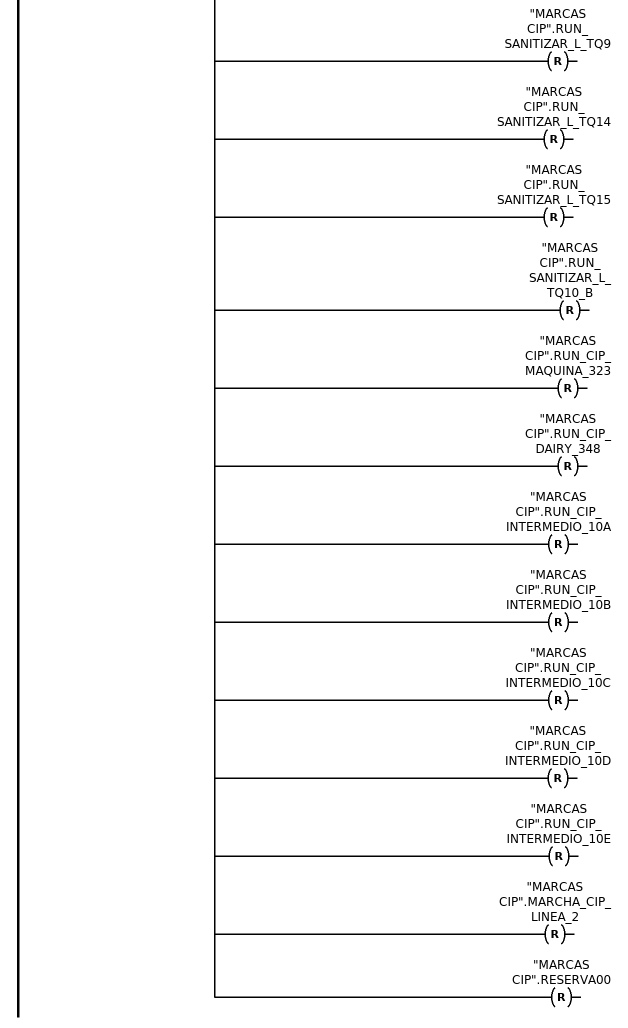
   RUNG wire#powerrail
      Contact( "PASOS CIP L2".paso_20_vaciado_tanque )
      Contact( "Tag_795" )
      wire#w1
      R_Coil( "PASOS CIP L2".paso_20_vaciado_tanque )
   END_RUNG
   RUNG wire#w1
      R_Coil( "MARCAS CIP".RUN_CIP_TANQUE_5 )
   END_RUNG
   RUNG wire#w1
      R_Coil( "MARCAS CIP".RUN_CIP_TANQUE_6 )
   END_RUNG
   RUNG wire#w1
      R_Coil( "MARCAS CIP".RUN_CIP_TQ14_15_FLAN )
   END_RUNG
   RUNG wire#w1
      R_Coil( "MARCAS CIP".RUN_CIP_FLAN_PAS2500 )
   END_RUNG
   RUNG wire#w1
      R_Coil( "MARCAS CIP".RUN_CIP_L_HORNO_VIEJO )
   END_RUNG
   RUNG wire#w1
      R_Coil( "MARCAS CIP".RUN_CIP_L_HORNO_PUDIN )
   END_RUNG
   RUNG wire#w1
      R_Coil( "MARCAS CIP".RUN_CIP_L_HORNO_BA1 )
   END_RUNG
   RUNG wire#w1
      R_Coil( "MARCAS CIP".RUN_CIP_HUEVO_A_FLAN )
   END_RUNG
   RUNG wire#w1
      R_Coil( "MARCAS CIP".RUN_CIP_TANQUE_7 )
   END_RUNG
   RUNG wire#w1
      R_Coil( "MARCAS CIP".RUN_CIP_TANQUE_8 )
   END_RUNG
   RUNG wire#w1
      R_Coil( "MARCAS CIP".RUN_CIP_TANQUE_9 )
   END_RUNG
   RUNG wire#w1
      R_Coil( "MARCAS CIP".RUN_CIP_TANQUE_10 )
   END_RUNG
   RUNG wire#w1
      R_Coil( "MARCAS CIP".RUN_CIP_L_DOSIF_TQ_10 )
   END_RUNG
   RUNG wire#w1
      R_Coil( "MARCAS CIP".RUN_CIP_DOSIF_NATILL )
   END_RUNG
   RUNG wire#w1
      R_Coil( "MARCAS CIP".RUN_CIP_DOSIF_VARIOS )
   END_RUNG
   RUNG wire#w1
      R_Coil( "MARCAS CIP".RUN_CIP_DAIRY_321 )
   END_RUNG
   RUNG wire#w1
      R_Coil( "MARCAS CIP".RUN_CIP_TQ_QUESO_FLAN )
   END_RUNG
   RUNG wire#w1
      R_Coil( "MARCAS CIP".RUN_CIP_L_RET_FLAN_TQ5_6 )
   END_RUNG
   RUNG wire#w1
      R_Coil( "MARCAS CIP".RUN_CIP_L_RECIR_TQ_QUESO )
   END_RUNG
   RUNG wire#w1
      R_Coil( "MARCAS CIP".RUN_CIP_TQ_MEZCL_ARROZ )
   END_RUNG
   RUNG wire#w1
      R_Coil( "MARCAS CIP".RUN_CIP_MAQUINA_GELATINA )
   END_RUNG
   RUNG wire#w1
      R_Coil( "MARCAS CIP".RUN_CIP_M_GELATINA_ULMA )
   END_RUNG
   RUNG wire#w1
      R_Coil( "MARCAS CIP".RUN_CIP_L_CLARA_TARTAS )
   END_RUNG
   RUNG wire#w1
      R_Coil( "MARCAS CIP".RUN_CIP_TANQUE_14 )
   END_RUNG
   RUNG wire#w1
      R_Coil( "MARCAS CIP".RUN_CIP_TANQUE_15 )
   END_RUNG
   RUNG wire#w1
      R_Coil( "MARCAS CIP".RUN_CIP_TANQUE_10_B )
   END_RUNG
   RUNG wire#w1
      R_Coil( "MARCAS CIP".RUN_CIP_TANQUE_10D )
   END_RUNG
   RUNG wire#w1
      R_Coil( "MARCAS CIP".RUN_CIP_TANQUE_10E )
   END_RUNG
   RUNG wire#w1
      R_Coil( "MARCAS CIP".RUN_CIP_TANQUE_10_C )
   END_RUNG
   RUNG wire#w1
      R_Coil( "MARCAS CIP".RUN_CIP_L_TQ14_15_LLEN )
   END_RUNG
   RUNG wire#w1
      R_Coil( "MARCAS CIP".RUN_CIP_L_CUBOS_YOGUR )
   END_RUNG
   RUNG wire#w1
      R_Coil( "MARCAS CIP".RUN_SANITIZAR_L_TQ7 )
   END_RUNG
   RUNG wire#w1
      R_Coil( "MARCAS CIP".RUN_SANITIZAR_L_TQ8 )
   END_RUNG
   RUNG wire#w1
      R_Coil( "MARCAS CIP".RUN_SANITIZAR_L_TQ9 )
   END_RUNG
   RUNG wire#w1
      R_Coil( "MARCAS CIP".RUN_SANITIZAR_L_TQ14 )
   END_RUNG
   RUNG wire#w1
      R_Coil( "MARCAS CIP".RUN_SANITIZAR_L_TQ15 )
   END_RUNG
   RUNG wire#w1
      R_Coil( "MARCAS CIP".RUN_SANITIZAR_L_TQ10_B )
   END_RUNG
   RUNG wire#w1
      R_Coil( "MARCAS CIP".RUN_CIP_MAQUINA_323 )
   END_RUNG
   RUNG wire#w1
      R_Coil( "MARCAS CIP".RUN_CIP_DAIRY_348 )
   END_RUNG
   RUNG wire#w1
      R_Coil( "MARCAS CIP".RUN_CIP_INTERMEDIO_10A )
   END_RUNG
   RUNG wire#w1
      R_Coil( "MARCAS CIP".RUN_CIP_INTERMEDIO_10B )
   END_RUNG
   RUNG wire#w1
      R_Coil( "MARCAS CIP".RUN_CIP_INTERMEDIO_10C )
   END_RUNG
   RUNG wire#w1
      R_Coil( "MARCAS CIP".RUN_CIP_INTERMEDIO_10D )
   END_RUNG
   RUNG wire#w1
      R_Coil( "MARCAS CIP".RUN_CIP_INTERMEDIO_10E )
   END_RUNG
   RUNG wire#w1
      R_Coil( "MARCAS CIP".MARCHA_CIP_LINEA_2 )
   END_RUNG
   RUNG wire#w1
      R_Coil( "MARCAS CIP".RESERVA00 )
   END_RUNG
   // the same network as SCL:
   #_w1 := "PASOS CIP L2".paso_20_vaciado_tanque AND "Tag_795";
   IF #_w1 THEN
       "PASOS CIP L2".paso_20_vaciado_tanque := FALSE;
       "MARCAS CIP".RUN_CIP_TANQUE_5 := FALSE;
       "MARCAS CIP".RUN_CIP_TANQUE_6 := FALSE;
       "MARCAS CIP".RUN_CIP_TQ14_15_FLAN := FALSE;
       "MARCAS CIP".RUN_CIP_FLAN_PAS2500 := FALSE;
       "MARCAS CIP".RUN_CIP_L_HORNO_VIEJO := FALSE;
       "MARCAS CIP".RUN_CIP_L_HORNO_PUDIN := FALSE;
       "MARCAS CIP".RUN_CIP_L_HORNO_BA1 := FALSE;
       "MARCAS CIP".RUN_CIP_HUEVO_A_FLAN := FALSE;
       "MARCAS CIP".RUN_CIP_TANQUE_7 := FALSE;
       "MARCAS CIP".RUN_CIP_TANQUE_8 := FALSE;
       "MARCAS CIP".RUN_CIP_TANQUE_9 := FALSE;
       "MARCAS CIP".RUN_CIP_TANQUE_10 := FALSE;
       "MARCAS CIP".RUN_CIP_L_DOSIF_TQ_10 := FALSE;
       "MARCAS CIP".RUN_CIP_DOSIF_NATILL := FALSE;
       "MARCAS CIP".RUN_CIP_DOSIF_VARIOS := FALSE;
       "MARCAS CIP".RUN_CIP_DAIRY_321 := FALSE;
       "MARCAS CIP".RUN_CIP_TQ_QUESO_FLAN := FALSE;
       "MARCAS CIP".RUN_CIP_L_RET_FLAN_TQ5_6 := FALSE;
       "MARCAS CIP".RUN_CIP_L_RECIR_TQ_QUESO := FALSE;
       "MARCAS CIP".RUN_CIP_TQ_MEZCL_ARROZ := FALSE;
       "MARCAS CIP".RUN_CIP_MAQUINA_GELATINA := FALSE;
       "MARCAS CIP".RUN_CIP_M_GELATINA_ULMA := FALSE;
       "MARCAS CIP".RUN_CIP_L_CLARA_TARTAS := FALSE;
       "MARCAS CIP".RUN_CIP_TANQUE_14 := FALSE;
       "MARCAS CIP".RUN_CIP_TANQUE_15 := FALSE;
       "MARCAS CIP".RUN_CIP_TANQUE_10_B := FALSE;
       "MARCAS CIP".RUN_CIP_TANQUE_10D := FALSE;
       "MARCAS CIP".RUN_CIP_TANQUE_10E := FALSE;
       "MARCAS CIP".RUN_CIP_TANQUE_10_C := FALSE;
       "MARCAS CIP".RUN_CIP_L_TQ14_15_LLEN := FALSE;
       "MARCAS CIP".RUN_CIP_L_CUBOS_YOGUR := FALSE;
       "MARCAS CIP".RUN_SANITIZAR_L_TQ7 := FALSE;
       "MARCAS CIP".RUN_SANITIZAR_L_TQ8 := FALSE;
       "MARCAS CIP".RUN_SANITIZAR_L_TQ9 := FALSE;
       "MARCAS CIP".RUN_SANITIZAR_L_TQ14 := FALSE;
       "MARCAS CIP".RUN_SANITIZAR_L_TQ15 := FALSE;
       "MARCAS CIP".RUN_SANITIZAR_L_TQ10_B := FALSE;
       "MARCAS CIP".RUN_CIP_MAQUINA_323 := FALSE;
       "MARCAS CIP".RUN_CIP_DAIRY_348 := FALSE;
       "MARCAS CIP".RUN_CIP_INTERMEDIO_10A := FALSE;
       "MARCAS CIP".RUN_CIP_INTERMEDIO_10B := FALSE;
       "MARCAS CIP".RUN_CIP_INTERMEDIO_10C := FALSE;
       "MARCAS CIP".RUN_CIP_INTERMEDIO_10D := FALSE;
       "MARCAS CIP".RUN_CIP_INTERMEDIO_10E := FALSE;
       "MARCAS CIP".MARCHA_CIP_LINEA_2 := FALSE;
       "MARCAS CIP".RESERVA00 := FALSE;
   END_IF;
END_REGION

REGION Network 64: Variable prvisional
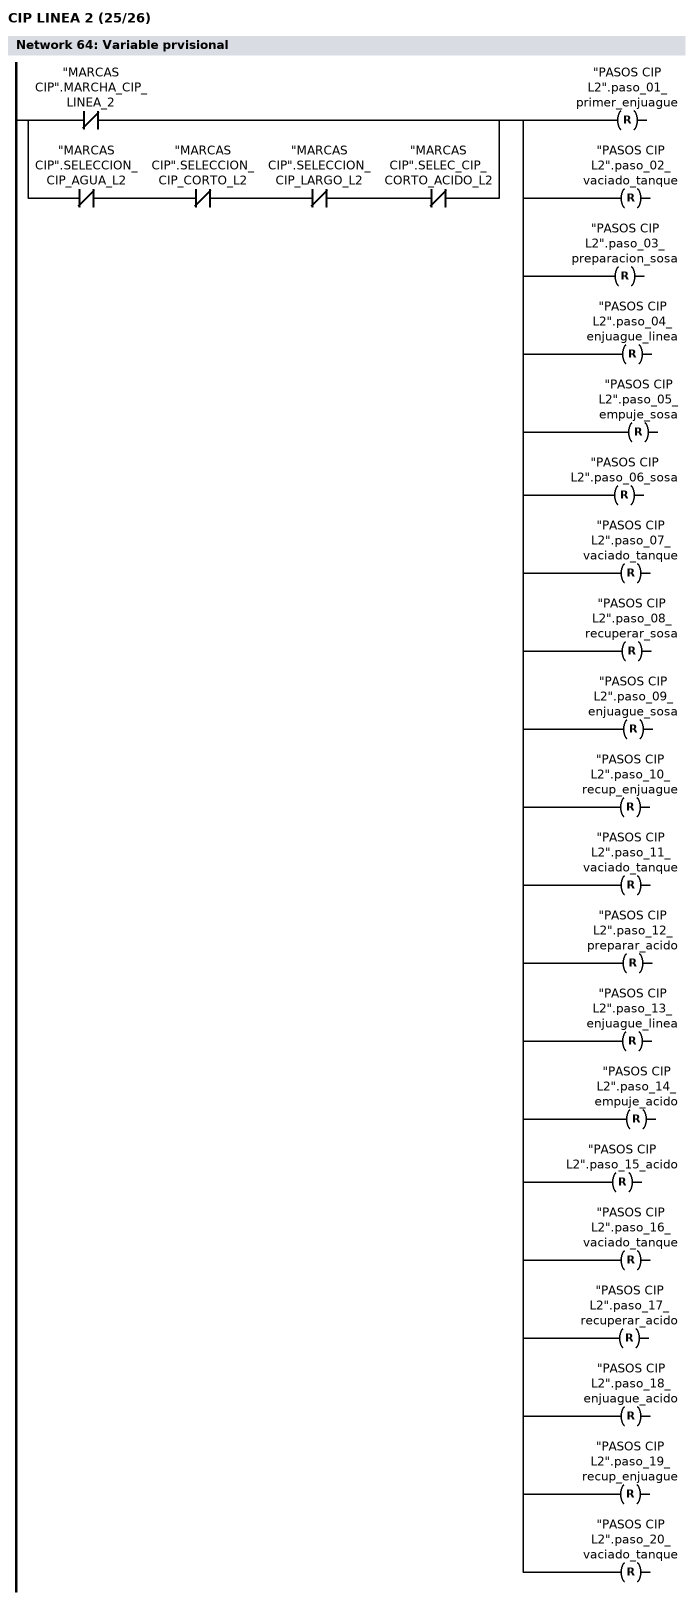
   RUNG wire#powerrail
      I_Contact( "MARCAS CIP".MARCHA_CIP_LINEA_2 )
      wire#w1
      R_Coil( "PASOS CIP L2".paso_01_primer_enjuague )
   END_RUNG
   RUNG wire#powerrail
      I_Contact( "MARCAS CIP".SELECCION_CIP_AGUA_L2 )
      I_Contact( "MARCAS CIP".SELECCION_CIP_CORTO_L2 )
      I_Contact( "MARCAS CIP".SELECCION_CIP_LARGO_L2 )
      I_Contact( "MARCAS CIP".SELEC_CIP_CORTO_ACIDO_L2 )
   END_RUNG wire#w1
   RUNG wire#w1
      R_Coil( "PASOS CIP L2".paso_02_vaciado_tanque )
   END_RUNG
   RUNG wire#w1
      R_Coil( "PASOS CIP L2".paso_03_preparacion_sosa )
   END_RUNG
   RUNG wire#w1
      R_Coil( "PASOS CIP L2".paso_04_enjuague_linea )
   END_RUNG
   RUNG wire#w1
      R_Coil( "PASOS CIP L2".paso_05_empuje_sosa )
   END_RUNG
   RUNG wire#w1
      R_Coil( "PASOS CIP L2".paso_06_sosa )
   END_RUNG
   RUNG wire#w1
      R_Coil( "PASOS CIP L2".paso_07_vaciado_tanque )
   END_RUNG
   RUNG wire#w1
      R_Coil( "PASOS CIP L2".paso_08_recuperar_sosa )
   END_RUNG
   RUNG wire#w1
      R_Coil( "PASOS CIP L2".paso_09_enjuague_sosa )
   END_RUNG
   RUNG wire#w1
      R_Coil( "PASOS CIP L2".paso_10_recup_enjuague )
   END_RUNG
   RUNG wire#w1
      R_Coil( "PASOS CIP L2".paso_11_vaciado_tanque )
   END_RUNG
   RUNG wire#w1
      R_Coil( "PASOS CIP L2".paso_12_preparar_acido )
   END_RUNG
   RUNG wire#w1
      R_Coil( "PASOS CIP L2".paso_13_enjuague_linea )
   END_RUNG
   RUNG wire#w1
      R_Coil( "PASOS CIP L2".paso_14_empuje_acido )
   END_RUNG
   RUNG wire#w1
      R_Coil( "PASOS CIP L2".paso_15_acido )
   END_RUNG
   RUNG wire#w1
      R_Coil( "PASOS CIP L2".paso_16_vaciado_tanque )
   END_RUNG
   RUNG wire#w1
      R_Coil( "PASOS CIP L2".paso_17_recuperar_acido )
   END_RUNG
   RUNG wire#w1
      R_Coil( "PASOS CIP L2".paso_18_enjuague_acido )
   END_RUNG
   RUNG wire#w1
      R_Coil( "PASOS CIP L2".paso_19_recup_enjuague )
   END_RUNG
   RUNG wire#w1
      R_Coil( "PASOS CIP L2".paso_20_vaciado_tanque )
   END_RUNG
   // the same network as SCL:
   IF NOT "MARCAS CIP".MARCHA_CIP_LINEA_2 OR (NOT "MARCAS CIP".SELECCION_CIP_AGUA_L2 AND NOT "MARCAS CIP".SELECCION_CIP_CORTO_L2 AND NOT "MARCAS CIP".SELECCION_CIP_LARGO_L2 AND NOT "MARCAS CIP".SELEC_CIP_CORTO_ACIDO_L2) THEN
       "PASOS CIP L2".paso_01_primer_enjuague := FALSE;
       "PASOS CIP L2".paso_02_vaciado_tanque := FALSE;
       "PASOS CIP L2".paso_03_preparacion_sosa := FALSE;
       "PASOS CIP L2".paso_04_enjuague_linea := FALSE;
       "PASOS CIP L2".paso_05_empuje_sosa := FALSE;
       "PASOS CIP L2".paso_06_sosa := FALSE;
       "PASOS CIP L2".paso_07_vaciado_tanque := FALSE;
       "PASOS CIP L2".paso_08_recuperar_sosa := FALSE;
       "PASOS CIP L2".paso_09_enjuague_sosa := FALSE;
       "PASOS CIP L2".paso_10_recup_enjuague := FALSE;
       "PASOS CIP L2".paso_11_vaciado_tanque := FALSE;
       "PASOS CIP L2".paso_12_preparar_acido := FALSE;
       "PASOS CIP L2".paso_13_enjuague_linea := FALSE;
       "PASOS CIP L2".paso_14_empuje_acido := FALSE;
       "PASOS CIP L2".paso_15_acido := FALSE;
       "PASOS CIP L2".paso_16_vaciado_tanque := FALSE;
       "PASOS CIP L2".paso_17_recuperar_acido := FALSE;
       "PASOS CIP L2".paso_18_enjuague_acido := FALSE;
       "PASOS CIP L2".paso_19_recup_enjuague := FALSE;
       "PASOS CIP L2".paso_20_vaciado_tanque := FALSE;
   END_IF;
END_REGION

REGION Network 65
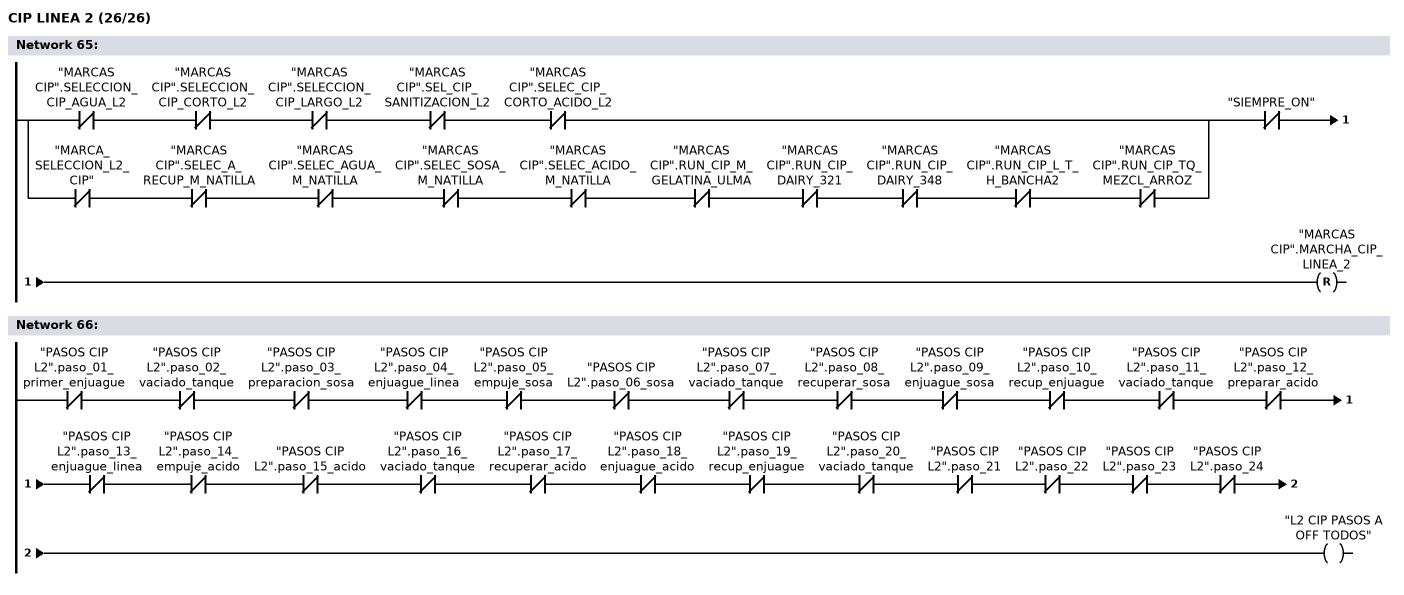
   RUNG wire#powerrail
      I_Contact( "MARCAS CIP".SELECCION_CIP_AGUA_L2 )
      I_Contact( "MARCAS CIP".SELECCION_CIP_CORTO_L2 )
      I_Contact( "MARCAS CIP".SELECCION_CIP_LARGO_L2 )
      I_Contact( "MARCAS CIP".SEL_CIP_SANITIZACION_L2 )
      I_Contact( "MARCAS CIP".SELEC_CIP_CORTO_ACIDO_L2 )
      wire#w1
      I_Contact( "SIEMPRE_ON" )
      R_Coil( "MARCAS CIP".MARCHA_CIP_LINEA_2 )
   END_RUNG
   RUNG wire#powerrail
      I_Contact( "MARCA_SELECCION_L2_CIP" )
      I_Contact( "MARCAS CIP".SELEC_A_RECUP_M_NATILLA )
      I_Contact( "MARCAS CIP".SELEC_AGUA_M_NATILLA )
      I_Contact( "MARCAS CIP".SELEC_SOSA_M_NATILLA )
      I_Contact( "MARCAS CIP".SELEC_ACIDO_M_NATILLA )
      I_Contact( "MARCAS CIP".RUN_CIP_M_GELATINA_ULMA )
      I_Contact( "MARCAS CIP".RUN_CIP_DAIRY_321 )
      I_Contact( "MARCAS CIP".RUN_CIP_DAIRY_348 )
      I_Contact( "MARCAS CIP".RUN_CIP_L_T_H_BANCHA2 )
      I_Contact( "MARCAS CIP".RUN_CIP_TQ_MEZCL_ARROZ )
   END_RUNG wire#w1
   // the same network as SCL:
   IF ((NOT "MARCAS CIP".SELECCION_CIP_AGUA_L2 AND NOT "MARCAS CIP".SELECCION_CIP_CORTO_L2 AND NOT "MARCAS CIP".SELECCION_CIP_LARGO_L2 AND NOT "MARCAS CIP".SEL_CIP_SANITIZACION_L2 AND NOT "MARCAS CIP".SELEC_CIP_CORTO_ACIDO_L2) OR (NOT "MARCA_SELECCION_L2_CIP" AND NOT "MARCAS CIP".SELEC_A_RECUP_M_NATILLA AND NOT "MARCAS CIP".SELEC_AGUA_M_NATILLA AND NOT "MARCAS CIP".SELEC_SOSA_M_NATILLA AND NOT "MARCAS CIP".SELEC_ACIDO_M_NATILLA AND NOT "MARCAS CIP".RUN_CIP_M_GELATINA_ULMA AND NOT "MARCAS CIP".RUN_CIP_DAIRY_321 AND NOT "MARCAS CIP".RUN_CIP_DAIRY_348 AND NOT "MARCAS CIP".RUN_CIP_L_T_H_BANCHA2 AND NOT "MARCAS CIP".RUN_CIP_TQ_MEZCL_ARROZ)) AND NOT "SIEMPRE_ON" THEN
       "MARCAS CIP".MARCHA_CIP_LINEA_2 := FALSE;
   END_IF;
END_REGION

REGION Network 66
   RUNG wire#powerrail
      I_Contact( "PASOS CIP L2".paso_01_primer_enjuague )
      I_Contact( "PASOS CIP L2".paso_02_vaciado_tanque )
      I_Contact( "PASOS CIP L2".paso_03_preparacion_sosa )
      I_Contact( "PASOS CIP L2".paso_04_enjuague_linea )
      I_Contact( "PASOS CIP L2".paso_05_empuje_sosa )
      I_Contact( "PASOS CIP L2".paso_06_sosa )
      I_Contact( "PASOS CIP L2".paso_07_vaciado_tanque )
      I_Contact( "PASOS CIP L2".paso_08_recuperar_sosa )
      I_Contact( "PASOS CIP L2".paso_09_enjuague_sosa )
      I_Contact( "PASOS CIP L2".paso_10_recup_enjuague )
      I_Contact( "PASOS CIP L2".paso_11_vaciado_tanque )
      I_Contact( "PASOS CIP L2".paso_12_preparar_acido )
      I_Contact( "PASOS CIP L2".paso_13_enjuague_linea )
      I_Contact( "PASOS CIP L2".paso_14_empuje_acido )
      I_Contact( "PASOS CIP L2".paso_15_acido )
      I_Contact( "PASOS CIP L2".paso_16_vaciado_tanque )
      I_Contact( "PASOS CIP L2".paso_17_recuperar_acido )
      I_Contact( "PASOS CIP L2".paso_18_enjuague_acido )
      I_Contact( "PASOS CIP L2".paso_19_recup_enjuague )
      I_Contact( "PASOS CIP L2".paso_20_vaciado_tanque )
      I_Contact( "PASOS CIP L2".paso_21 )
      I_Contact( "PASOS CIP L2".paso_22 )
      I_Contact( "PASOS CIP L2".paso_23 )
      I_Contact( "PASOS CIP L2".paso_24 )
      Coil( "L2 CIP PASOS A OFF TODOS" )
   END_RUNG
   // the same network as SCL:
   "L2 CIP PASOS A OFF TODOS" := NOT "PASOS CIP L2".paso_01_primer_enjuague AND NOT "PASOS CIP L2".paso_02_vaciado_tanque AND NOT "PASOS CIP L2".paso_03_preparacion_sosa AND NOT "PASOS CIP L2".paso_04_enjuague_linea AND NOT "PASOS CIP L2".paso_05_empuje_sosa AND NOT "PASOS CIP L2".paso_06_sosa AND NOT "PASOS CIP L2".paso_07_vaciado_tanque AND NOT "PASOS CIP L2".paso_08_recuperar_sosa AND NOT "PASOS CIP L2".paso_09_enjuague_sosa AND NOT "PASOS CIP L2".paso_10_recup_enjuague AND NOT "PASOS CIP L2".paso_11_vaciado_tanque AND NOT "PASOS CIP L2".paso_12_preparar_acido AND NOT "PASOS CIP L2".paso_13_enjuague_linea AND NOT "PASOS CIP L2".paso_14_empuje_acido AND NOT "PASOS CIP L2".paso_15_acido AND NOT "PASOS CIP L2".paso_16_vaciado_tanque AND NOT "PASOS CIP L2".paso_17_recuperar_acido AND NOT "PASOS CIP L2".paso_18_enjuague_acido AND NOT "PASOS CIP L2".paso_19_recup_enjuague AND NOT "PASOS CIP L2".paso_20_vaciado_tanque AND NOT "PASOS CIP L2".paso_21 AND NOT "PASOS CIP L2".paso_22 AND NOT "PASOS CIP L2".paso_23 AND NOT "PASOS CIP L2".paso_24;
END_REGION
END_FUNCTION
